PROGRAM P_Inputs
VAR
	fbJoystickWinch 				: FB_JoystickInputScaling;
	fbJoystickCyl 					: FB_JoystickInputScaling;
	fbJoystickRot 					: FB_JoystickInputScaling;
	fbYokeInputScaling 				: FB_YokeInputScaling;
	fbWinchPosition 				: FB_Encoder;
	fbPressureSupply 				: FB_AnalogInputScaling;
	fbPressureReturn 				: FB_AnalogInputScaling;
	fbPressureWinch_A_Input 		: FB_AnalogInputScaling;
	fbPressureWinch_B_Output		: FB_AnalogInputScaling;
	eStatus						    : E_Status;
END_VAR

fbJoystickWinch(
	bEnable := G_IO.bManualSwtich OR G_IO.bAutoSwtich,
	nRawInput := G_IO.fJoyYraw,
	stJoystickInputScaling := G_Parameters.stParam.stJoystickInputScalingY,
	fNormalizedOutput => G_Sensors.fJoystickNormalizedY
);

fbJoystickRot(
	bEnable := G_IO.bManualSwtich,
	nRawInput := G_IO.fJoyZraw,
	stJoystickInputScaling := G_Parameters.stParam.stJoystickInputScalingZ,
	fNormalizedOutput => G_Sensors.fJoystickNormalizedZ
);

fbYokeInputScaling(
	bEnable := G_IO.bManualSwtich,
	nRawInput := G_IO.fYoke,
	stYokeInputScaling := G_Parameters.stParam.stYokeInputScaling,
	fNormalizedOutput => G_Sensors.fYokeNormalizedFeedback
);

fbWinchPosition (
	nRawInput := G_IO.nWinchEncoderValue, 
	fEncoderOffset := G_Parameters.stParam.fWinchEncoderOffset,
	fPosition => G_Sensors.fWinchEncoderPosition
);

fbPressureSupply(
	nRawInput := G_IO.fPressureSupply,
	stAnalogInputScaling := G_Parameters.stParam.stPressureSensorScaling400bar,
	fOutput => G_Sensors.fPressureSupply
);

fbPressureReturn(
	nRawInput := G_IO.fPressureReturn,
	stAnalogInputScaling := G_Parameters.stParam.stPressureSensorScaling40bar,
	fOutput => G_Sensors.fPressureReturn
);

fbPressureWinch_A_Input(
	nRawInput := G_IO.fPressureWinchA,
	stAnalogInputScaling := G_Parameters.stParam.stPressureSensorScaling400bar,
	fOutput => G_Sensors.fPressureWinchA
);

// I deed a Thng Nils
fbPressureWinch_B_Output(
	nRawInput := G_IO.fPressureCylinderA,
	stAnalogInputScaling := G_Parameters.stParam.stPressureSensorScaling400bar,
	fOutput => G_Sensors.fPressureWinchB
);

G_Sensors.fDeltaPMotor := (G_Sensors.fPressureWinchB - G_Sensors.fPressureWinchA);

END_PROGRAM

(* stored: Version 1.1.0.1, ProductVersion 3.1.4024.12
   POU P_Inputs: Id {8b676dbd-393f-42d6-8803-330b6e90ab14}, SpecialFunc None *)
